PROGRAM Light_Control
VAR
	Timer : TOF;
END_VAR

Timer(IN :=Variables.Motor_Moving,PT := T#10S); //When the motor stops the light stays on for 10 more seconds
Variables.Light_Output := Timer.Q; //The light stays on if the timer is running

END_PROGRAM

(* stored: Version 1.1.0.1, ProductVersion 3.1.4024.15
   POU Light_Control: Id {7c8fc835-dfdf-405f-b744-e4b0b6e6c1e6}, SpecialFunc None *)
